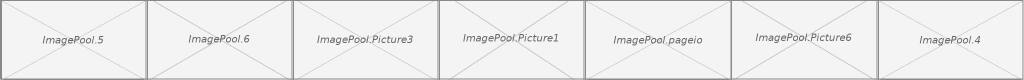
VISUALIZATION N_Footer_Line2  // 1024x80
    Image (1,0 145x80), input disabled if: Not bResetmanual2, image: ImagePool.5
        OnMouseDown: change screen: MAIN_LINE2
        OnMouseDown: execute { MAIN_LINE2.bModeAuto := TRUE; MAIN_LINE2.bModeManual := FALSE; }
    Image (147,-3 145x84), input disabled if: bResetAuto2, image: ImagePool.6
        OnMouseDown: change screen: N_JarSupply2
        OnMouseDown: execute { MAIN_LINE2.bModeManual := TRUE; MAIN_LINE2.bModeAuto := FALSE; }
    Image (293,-2 145x83), image: ImagePool.Picture3
        OnMouseClick: change screen: N_Setting_Line2
    Image (439,-10 145x96), image: ImagePool.Picture1
        OnMouseClick: change screen: N_Recipe_Line2
    Image (585,0 146x80), image: ImagePool.pageio
        OnMouseClick: change screen: N_PLC_I2
    Image (731,-6 146x87), image: ImagePool.Picture6
        OnMouseClick: change screen: N_Alarm_1
    Image (878,0 145x80), invisible if: GVL_OF_VU.bVN, input disabled if: GVL_OF_VU.bVN, image: ImagePool.3
        OnMouseDown: ChangeLanguage ChangeLanguage=vn
    Image (878,0 145x80), invisible if: not GVL_OF_VU.bVN, input disabled if: not GVL_OF_VU.bVN, image: ImagePool.4
        OnMouseDown: ChangeLanguage ChangeLanguage=eng
END_VISUALIZATION

(* stored: Version 1.1.0.1, ProductVersion 3.1.4024.12
   Visu N_Footer_Line2: Id {4fd3c67f-180e-4353-8e0d-c51a5e773251} *)
